PROGRAM StartVisu

VAR_INPUT
    NETID     : T_AmsNetId;
    PATHSTR   : T_MaxString;
    DIRNAME   : T_MaxString;
    COMNDLINE : T_MaxString;
    START     : BOOL;
    TMOUT     : TIME := DEFAULT_ADS_TIMEOUT;
END_VAR



VAR
END_VAR

END_PROGRAM

(* stored: Version 1.1.0.1, ProductVersion 3.1.4024.0
   POU StartVisu: Id {1c588346-da7f-4d04-bd3b-df15b94685cb}, SpecialFunc None *)
